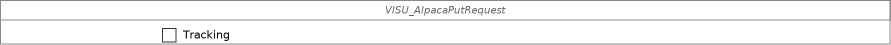
VISUALIZATION VISU_AlpacaPutTracking  // 891x45
VAR_IN_OUT
	stInstance : ST_AlpacaPutTracking;
END_VAR
    Frame (0,0 891x20)
        shows VISU_AlpacaPutRequest(stInstance := stInstance)
    Checkbox (160,25 121x20), "Tracking", variable: stInstance.i_bTracking
END_VISUALIZATION

(* stored: Version 1.1.0.1, ProductVersion 3.1.4024.12
   Visu VISU_AlpacaPutTracking: Id {2b41006b-9688-457a-86fe-2452611af7b5} *)
